(* PLC project PLC1, Unknown Unnamed 1 *)
(* stored: creationDateTime 2021-02-24T14:42:08, modificationDateTime 2024-08-19T11:14:29 *)

PROGRAM PLC3
  VAR_INPUT
    level : DINT;
  END_VAR
  VAR_OUTPUT
    pump : BOOL;
  END_VAR
  VAR
    low : BOOL;
    high : BOOL;
    low_3 : DINT := 0;
    high_3 : DINT := 10;
  END_VAR

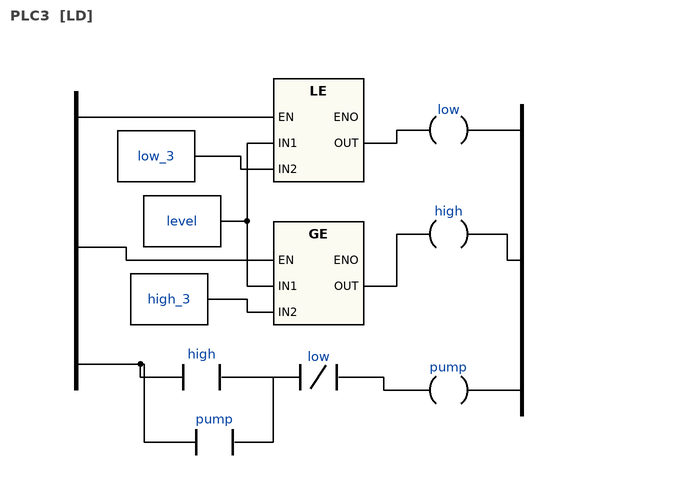
(* LD diagram, written out as Structured Text *)
high := level >= high_3;
low := level <= low_3;
pump := (high OR pump) AND NOT low;
END_PROGRAM

PROGRAM PLC2
  VAR_INPUT
    level : DINT;
  END_VAR
  VAR_OUTPUT
    request : BOOL;
  END_VAR
  VAR
    open_req : BOOL;
    close_req : BOOL;
    low_2 : DINT := 10;
    high_2 : DINT := 20;
  END_VAR

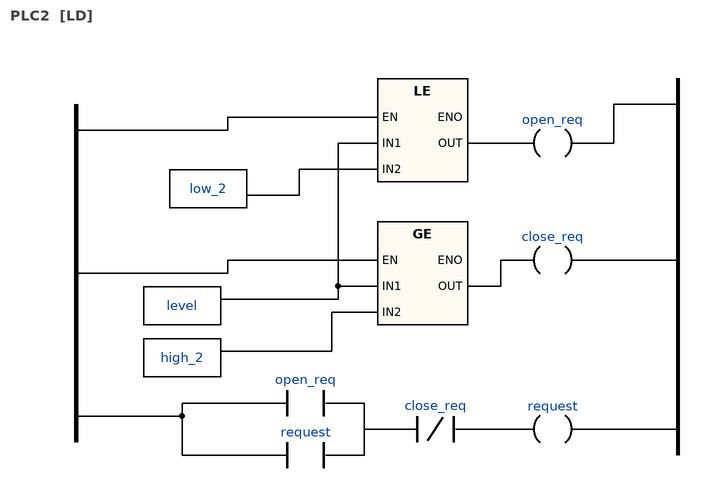
(* LD diagram, written out as Structured Text *)
close_req := level >= high_2;
open_req := level <= low_2;
request := (open_req OR request) AND NOT close_req;
END_PROGRAM

FUNCTION_BLOCK GE_0
  VAR_INPUT
    IN1 : DINT;
    IN2 : DINT;
  END_VAR
  VAR_OUTPUT
    OUT : BOOL;
  END_VAR
  VAR
    i : INT;
    exc : __SYSTEM.ExceptionCode;
  END_VAR

            __TRY
OUT:=FALSE;
IF IN1>=IN2 THEN
  OUT:=TRUE;
END_IF;
__CATCH(exc)
  i:=0;
  while i<5 do
    OUT:=TRUE;
  end_while;
__ENDTRY;
          
END_FUNCTION_BLOCK

(* IN1 *)
PROGRAM PLC1
  VAR_INPUT
    level : DINT;
    request : DINT;
    IN1 : BOOL;
  END_VAR
  VAR_OUTPUT
    pumps : BOOL;
    valve : BOOL;
    high : BOOL;
  END_VAR
  VAR
    close_req : BOOL;
    low : BOOL;
    open_req : BOOL;
    low_1 : DINT := 40;
    high_1 : DINT := 80;
    GE_00 : GE_0;
  END_VAR

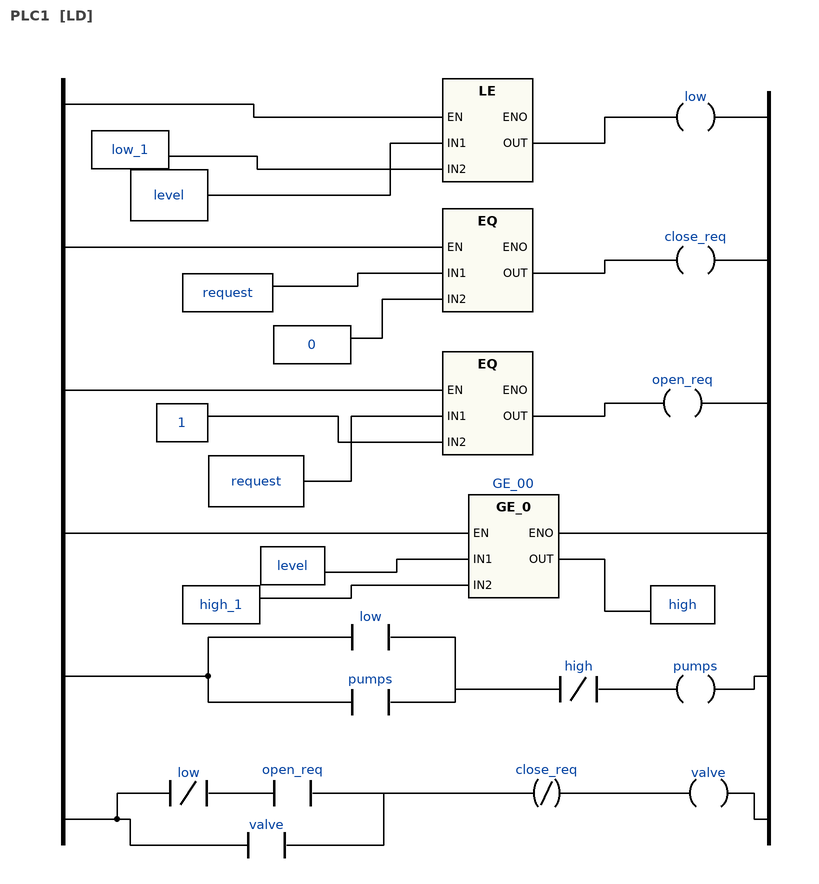
(* LD diagram, written out as Structured Text *)
low := level <= low_1;
close_req := request = 0;
pumps := (low OR pumps) AND NOT high;
valve := NOT low AND open_req OR valve;
open_req := request = 1;
close_req := NOT (NOT low AND open_req OR valve);
GE_00(IN1 := level, IN2 := high_1);
high := GE_00.OUT;
END_PROGRAM

CONFIGURATION Config0
  RESOURCE Res0 ON PLC
    TASK task0(INTERVAL := T#20ms, PRIORITY := 0);
    TASK task1(INTERVAL := T#20ms, PRIORITY := 0);
    TASK task2(INTERVAL := T#20ms, PRIORITY := 0);
    PROGRAM instance0 WITH task0 : PLC1;
    PROGRAM instance1 WITH task1 : PLC2;
    PROGRAM instance2 WITH task2 : PLC3;
  END_RESOURCE
END_CONFIGURATION
